FUNCTION_BLOCK EC_Scale (* Commands of Scale as output values, in timed phases: Idle=0, Tare=1, Measure=2 *)
  (* Standard: 61499-2 *)
  (* Version 0.1, 2026-09-28, Project contributors, AAU Smart Production Lab *)
  PACKAGE filling;
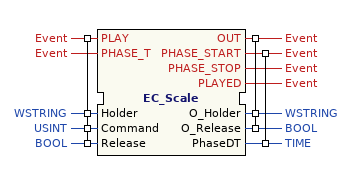
  EVENT_INPUT
    PLAY WITH Holder, Command, Release;
    PHASE_T;
  END_EVENT
  EVENT_OUTPUT
    OUT WITH O_Holder, O_Release;
    PHASE_START WITH PhaseDT;
    PHASE_STOP;
    PLAYED;
  END_EVENT
  VAR_INPUT
    Holder : WSTRING;
    Command : USINT;
    Release : BOOL;
  END_VAR
  VAR_OUTPUT
    O_Holder : WSTRING;
    O_Release : BOOL;
    PhaseDT : TIME;
  END_VAR
  VAR
    Phase : USINT;
    Timed : BOOL;
  END_VAR
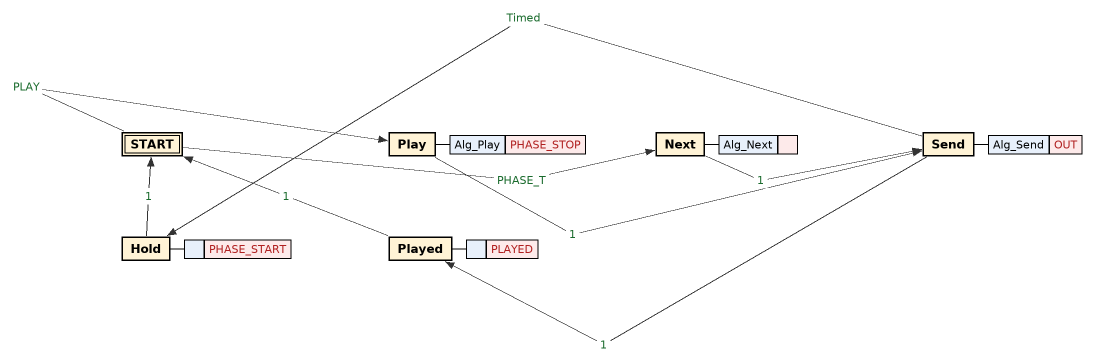
  EC_STATES
    START;
    Play : Alg_Play -> PHASE_STOP;
    Next : Alg_Next;
    Send : Alg_Send -> OUT;
    Hold : -> PHASE_START;
    Played : -> PLAYED;
  END_STATES
  EC_TRANSITIONS
    START TO Play := PLAY;
    START TO Next := PHASE_T;
    Play TO Send := 1;
    Next TO Send := 1;
    Send TO Hold := Timed;
    Send TO Played := 1;
    Hold TO START := 1;
    Played TO START := 1;
  END_TRANSITIONS
  ALGORITHM Alg_Play IN ST:
Phase := 0;
  END_ALGORITHM
  ALGORITHM Alg_Next IN ST:
Phase := Phase + 1;
  END_ALGORITHM
  ALGORITHM Alg_Send IN ST:
Timed := FALSE;
PhaseDT := T#0ms;
O_Holder := Holder;
O_Release := Release AND NOT Timed;
  END_ALGORITHM
END_FUNCTION_BLOCK
